// TwinCAT 3 PLC project PLC01
// ProgramVersion: 3.1.4024.0
// libraries:
//   Tc2_Standard, * (Beckhoff Automation GmbH)
//   Tc2_System, * (Beckhoff Automation GmbH)
//   Tc2_Utilities, * (Beckhoff Automation GmbH)
//   Tc3_Database, * (Beckhoff Automation GmbH)
//   Tc3_EventLogger, * (Beckhoff Automation GmbH)
//   Tc3_Module, * (Beckhoff Automation GmbH)
// project tree:
//   DUTs/ ST_Database.TcDUT
//   FBs/ FB_SQLMode_ExecuteCommandWithData.TcPOU, FB_SQLMode_ExecuteComandWithoutData.TcPOU, FB_SQLMode_ExecuteStoredProcedureWithoutData.TcPOU, FB_SQLMode_ExecuteStoredProcedureWithData.TcPOU
//   / PlcTask.TcTTO
//   POUs/ MAIN.TcPOU
//   POUs/PLC Mode/ PLC_Mode.TcPOU, PRG_CreateDatabasePlcMode.TcPOU, PRG_CreateTablePlcMode.TcPOU, PRG_DeleteRowDatabasePlcMode.TcPOU, PRG_ReadDatabasePlcMode.TcPOU, PRG_WriteDatabasePlcMode.TcPOU
//   POUs/SQL Mode/ PRG_CreateDatabaseSqlMode.TcPOU, PRG_CreateTableSqlMode.TcPOU, PRG_DeleteRowSqlMode.TcPOU, PRG_ReadDatabaseSqlMode.TcPOU, PRG_WriteDatabaseSqlMode.TcPOU, SQL_Mode.TcPOU
// real-time tasks:
//   TASK PlcTask: cycle T#10ms, priority 20, ADS port 350

CONFIGURATION PLC01
    RESOURCE PLC ON TwinCAT3
        TASK PlcTask(INTERVAL := T#10ms, PRIORITY := 20);
        PROGRAM MAIN WITH PlcTask : MAIN;
    END_RESOURCE
END_CONFIGURATION

// ---- DUTs/ST_Database.TcDUT
TYPE ST_Database :
STRUCT
	ID : T_ULARGE_INTEGER  ;	//IDENTITY
	Timestamp : DATE_AND_TIME ;	//TIMESTAMP
	recipe : STRING(51) ;		//NAME OF RECIPE
	parameter1 : LREAL ;		//PARAMETER 1
	parameter2 : LREAL ;		//PARAMETER 2
	parameter3 : LREAL ;		//PARAMETER 3
	parameter4 : LREAL ;		//PARAMETER 4
	parameter5 : LREAL ;		//PARAMETER 5
	parameter6 : LREAL ;		//PARAMETER 6
END_STRUCT
END_TYPE

// ---- POUs/MAIN.TcPOU
PROGRAM MAIN
VAR
END_VAR

PLC_Mode() ;

SQL_Mode();

END_PROGRAM

// ---- POUs/PLC Mode/PLC_Mode.TcPOU
PROGRAM PLC_Mode
VAR
END_VAR

PRG_CreateDatabasePlcMode();

PRG_CreateTablePlcMode();

PRG_DeleteRowDatabasePlcMode();

PRG_WriteDatabasePlcMode();

PRG_ReadDatabasePlcMode();

END_PROGRAM

// ---- POUs/PLC Mode/PRG_CreateDatabasePlcMode.TcPOU
PROGRAM PRG_CreateDatabasePlcMode
VAR
    fbPLCDBCreate : FB_PLCDBCreateEvt(sNetID := '', tTimeout := T#5S);
    stConfigDB    : T_DBConfig_MsSQL;
    hDBID         : UDINT ;
    tcMessage     : I_TcMessage;
	nState : INT ;	
	bCreateDatabase: BOOL;
	sMessage : STRING ;
END_VAR

stConfigDB.sProvider := 'SQLOLEDB' ;
stConfigDB.sServer:= 'DOUGLASC-NB01\SQLEXPRESS';
stConfigDB.sDatabase := 'MyDatabase123';
stConfigDB.bAuthentification := TRUE;
stConfigDB.sUserID := 'sa';
stConfigDB.sPassword := 'sa';

IF bCreateDatabase = TRUE THEN
	IF fbPLCDBCreate.Database(
		pDatabaseConfig:= ADR(stConfigDB),
		cbDatabaseConfig := SIZEOF(stConfigDB),
		bCreateXMLConfig := TRUE,
		pDBID := ADR(hDBID))
	THEN
		IF fbPLCDBCreate.bError THEN
			tcMessage := fbPLCDBCreate.ipTcResult;
			bCreateDatabase := FALSE ;
			sMessage := 'Error';
		ELSE
			bCreateDatabase := FALSE ;
			sMessage := 'OK';
		END_IF
	END_IF
END_IF

END_PROGRAM

// ---- POUs/PLC Mode/PRG_CreateTablePlcMode.TcPOU
PROGRAM PRG_CreateTablePlcMode
VAR
    fbPLCDBCreate	: FB_PLCDBCreateEvt(sNetID := '', tTimeout := T#5S);	//Bloco para criar a tabela
    ColumnInfo		: ARRAY [0..8] OF ST_ColumnInfo ;						//Estrutura com a tabela a ser criada
    tcMessage		: I_TcMessage;											//Variavel para tratamento das mensagens
	bCreateTable	: BOOL ; 												//Bit para criar tabela
	sError : STRING ;														//String com a mensagem de erro
END_VAR

(* Exemplos : 
ColumnInfo[0].sName := 'colBigInt';     ColumnInfo[0].eType := E_ColumnType.BigInt;     ColumnInfo[0].nLength := 8;     ColumnInfo[0].sProperty := 'IDENTITY(1,1)';
ColumnInfo[1].sName := 'colInteger';    ColumnInfo[1].eType := E_ColumnType.Integer;    ColumnInfo[1].nLength := 4;
ColumnInfo[2].sName := 'colSmallInt';   ColumnInfo[2].eType := E_ColumnType.SmallInt;   ColumnInfo[2].nLength := 2;
ColumnInfo[3].sName := 'colTinyInt';    ColumnInfo[3].eType := E_ColumnType.TinyInt;    ColumnInfo[3].nLength := 1;
ColumnInfo[4].sName := 'colBit';        ColumnInfo[4].eType := E_ColumnType.BIT_;       ColumnInfo[4].nLength := 1;
ColumnInfo[5].sName := 'colMoney';      ColumnInfo[5].eType := E_ColumnType.Money;      ColumnInfo[5].nLength := 8;
ColumnInfo[6].sName := 'colFloat';      ColumnInfo[6].eType := E_ColumnType.Float;      ColumnInfo[6].nLength := 8;
ColumnInfo[7].sName := 'colReal';       ColumnInfo[7].eType := E_ColumnType.REAL_;      ColumnInfo[7].nLength := 4;
ColumnInfo[8].sName := 'colDateTime';   ColumnInfo[8].eType := E_ColumnType.DateTime;   ColumnInfo[8].nLength := 4;
ColumnInfo[9].sName := 'colNText';      ColumnInfo[9].eType := E_ColumnType.NText;      ColumnInfo[9].nLength := 256;
ColumnInfo[10].sName := 'colNChar';     ColumnInfo[10].eType := E_ColumnType.NChar;     ColumnInfo[10].nLength := 10;
ColumnInfo[11].sName := 'colImage';     ColumnInfo[11].eType := E_ColumnType.Image;     ColumnInfo[11].nLength := 256;
ColumnInfo[12].sName := 'colNVarChar';  ColumnInfo[12].eType := E_ColumnType.NVarChar;  ColumnInfo[12].nLength := 50;
ColumnInfo[13].sName := 'colBinary';    ColumnInfo[13].eType := E_ColumnType.Binary;    ColumnInfo[13].nLength := 30;
ColumnInfo[14].sName := 'colVarBinary'; ColumnInfo[14].eType := E_ColumnType.VarBinary; ColumnInfo[14].nLength := 20;
*)

(* A criação das tabelas pode ser feita pelo código do PLC, mas também através da janela Sql Query Edition *)
(* Declaração da estrutura da tabela *)

ColumnInfo[0].sName := 'ID';     ColumnInfo[0].eType := E_ColumnType.BigInt;     ColumnInfo[0].nLength := 8;     ColumnInfo[0].sProperty := 'IDENTITY(1,1)';
ColumnInfo[1].sName := 'Timestamp';   ColumnInfo[1].eType := E_ColumnType.DateTime;   ColumnInfo[1].nLength := 4;
ColumnInfo[2].sName := 'recipe';  ColumnInfo[2].eType := E_ColumnType.NVarChar;  ColumnInfo[2].nLength := 50;
ColumnInfo[3].sName := 'parameter1';      ColumnInfo[3].eType := E_ColumnType.Float;      ColumnInfo[3].nLength := 8;
ColumnInfo[4].sName := 'parameter2';      ColumnInfo[4].eType := E_ColumnType.Float;      ColumnInfo[4].nLength := 8;
ColumnInfo[5].sName := 'parameter3';      ColumnInfo[5].eType := E_ColumnType.Float;      ColumnInfo[5].nLength := 8;
ColumnInfo[6].sName := 'parameter4';      ColumnInfo[6].eType := E_ColumnType.Float;      ColumnInfo[6].nLength := 8;
ColumnInfo[7].sName := 'parameter5';      ColumnInfo[7].eType := E_ColumnType.Float;      ColumnInfo[7].nLength := 8;
ColumnInfo[8].sName := 'parameter6';      ColumnInfo[8].eType := E_ColumnType.Float;      ColumnInfo[8].nLength := 8;

(* Para criar a tabela colocar a variavel bCreateTable em TRUE *)
(* To Create Table put the bCreateTable variable in TRUE *)
IF bCreateTable = TRUE THEN
	IF fbPLCDBCreate.Table(
		hDBID:= 1,
		sTableName:= 'TB_PLCMODE', 
		pTableCfg:= ADR(ColumnInfo), 
		cbTableCfg:= SIZEOF(ColumnInfo))
	THEN
		IF fbPLCDBCreate.bError THEN
			TcMessage:= fbPLCDBCreate.ipTcResult;
			sError := 'Erro'; 
		ELSE
			sError := 'OK';
		END_IF
	END_IF
	bCreateTable := FALSE ;	
END_IF

END_PROGRAM

// ---- POUs/PLC Mode/PRG_DeleteRowDatabasePlcMode.TcPOU
PROGRAM PRG_DeleteRowDatabasePlcMode
VAR
//Variáveis de conexão / Connection variables
	hDBID: UDINT := 1 ;							//DB ID
    sTableName: T_MaxString := 'TB_PLCMODE' ;	//Nome da Tabela / Table name

    fbPLCDBCmd		: FB_PLCDBCmdEvt(sNetID := '', tTimeout := T#5S);
    sCommandDelete  : STRING (1000);									//Comando SQL / SQL Command
    stParameter 	: ARRAY [1..1] OF ST_ExpParameter; 					//Parametros do comando SQL / Parameter SQL Command
    sRecipeName		: STRING(80) := 'recipe'; 							//Nome da receita a ser deletada / Recipe name to delete	
	bExecuteDelete 	: BOOL ;											//Executar delete / Execute delete	
	sMessageError	: STRING ;											//Mensagem de status / Status message
    tcMessageDelete	: I_TcMessage;										//
END_VAR

(***************************** CODE TO DELETE ONE ROW IN DATABASE             ***************************************)
(***************************** CODIGO PARA DELETAR UMA LINHA DO BANCO DE DADOS***************************************)

(* PARAMETER TO DELETE ONE RECIPE *)
(* PARAMETRO PARA DELETAR UMA RECEITA *)

stParameter[1].sParaName := 'sRecipeName';
stParameter[1].eParaType := E_ExpParameterType.STRING_;
stParameter[1].nParaSize := SIZEOF(sRecipeName);

(* SQL COMMAND TO DELETE A LINE THAT CONTAINS THE NAME DEFINED IN THE sRecipeName VARIABLE *)
(* COMANDO SQL PARA DELETAR UMA LINHA QUE CONTENHA O NOME DEFINIDO NA VARIAVEL sRecipeName *)
 sCommandDelete := 'DELETE FROM TB_PLCMODE WHERE recipe = {sRecipeName} ' ;
 
 
(* EXECUTE COMMAND TO DELETE THE ROW*)
(* EXECUTA COMANDO PARA DELETAR A LINHA *)
IF bExecuteDelete THEN

	IF fbPLCDBCmd.Execute(
		hDBID:= 1,
		pExpression:= ADR(sCommandDelete),
		cbExpression:= SIZEOF(sCommandDelete),
		pData:= ADR(sRecipeName),
		cbData:= SIZEOF(sRecipeName),
		pParameter:= ADR(stParameter),
		cbParameter:= SIZEOF(stParameter))				
	THEN	
		IF fbPLCDBCmd.bError THEN
			sMessageError := 'ERROR';
			bExecuteDelete := FALSE ;			
			tcMessageDelete := fbPLCDBCmd.ipTcResult;
		ELSE
			sMessageError := 'OK';
			bExecuteDelete := FALSE ;
		END_IF
	END_IF
END_IF

END_PROGRAM

// ---- POUs/PLC Mode/PRG_WriteDatabasePlcMode.TcPOU
PROGRAM PRG_WriteDatabasePlcMode
VAR
	hDBID: UDINT := 1 ;							//DB ID
    sTableName: T_MaxString := 'TB_PLCMODE' ;	//NOME DA TABELA / TABLE NAME / NOMBRE DA TABLA

//ESCREVER NO BANCO DE DADOS / WRITE DO DATABASE / ESCRIBIR EN LA BASE DE DATOS 
    fbPLCDBWrite    :	FB_PLCDBWriteEvt(sNetID := '', tTimeout := T#5S);//
    DataToDB 		:	ST_Database;									 //ESTRUTURA A ESCRITA NO BANCO / STRUCT TO SEND TO DATABASE
    ColumnNames     :	ARRAY[0..8] OF STRING(50);						 //ESTRUTURA COM O NOME DAS COLUNAS / STRUCT WITH COLLUNS NAME
    systime         :	GETSYSTEMTIME;									 //DATA E HORA DO  SISTEMA / DATE TIME OF SYSTEM
    currentTime     :	T_FILETIME;										 //
    tcMessage_Write :	I_TcMessage;									 //
	
	bWriteValues : BOOL ;	
	sMessage : STRING ;
	iRecipeNumerForTest : INT ;

END_VAR

//NOME DAS COLUNAS DA TABELA / NAME OF THE TABLE COLUMNS/
ColumnNames[0] := 'ID';
ColumnNames[1] := 'Timestamp';
ColumnNames[2] := 'recipe';
ColumnNames[3] := 'parameter1';
ColumnNames[4] := 'parameter2';
ColumnNames[5] := 'parameter3';
ColumnNames[6] := 'parameter4';
ColumnNames[7] := 'parameter5';
ColumnNames[8] := 'parameter6';

(* Logica de teste apenas para gerar dados para gravar no banco *)

systime(timeLoDw => currentTime.dwLowDateTime, timeHiDW => currentTime.dwHighDateTime );


(* SIMULATE VALUES TO WRITE TO DATABASE *)
IF bWriteValues THEN
	
//Simulacao de valores 
	DataToDB.Timestamp  := FILETIME_TO_DT(currentTime);;
	DataToDB.recipe     := CONCAT ('recipe', TO_STRING(iRecipeNumerForTest)) ;
	DataToDB.parameter1 := DataToDB.parameter1 + 10;
	DataToDB.parameter2 := DataToDB.parameter2 + 10;
	DataToDB.parameter3	:= DataToDB.parameter3 + 10 ;
	DataToDB.parameter4 := DataToDB.parameter4 + 10 ;
	DataToDB.parameter5 := DataToDB.parameter5 + 10 ;
	DataToDB.parameter6 := DataToDB.parameter6 + 10 ;

	
END_IF
	
/////////////////////////////// Chamada da função de escrita
IF bWriteValues THEN
	IF fbPLCDBWrite.WriteStruct(
		hDBID:= hDBID, 
		sTableName:= sTableName, 
		pRecord:= ADR(DataToDB), 
		cbRecord:= SIZEOF(DataToDB), 
		pColumnNames:= ADR(ColumnNames) , 
		cbColumnNames:= SIZEOF(ColumnNames))
	THEN
		IF fbPLCDBWrite.bError THEN
			tcMessage_Write := fbPLCDBWrite.ipTcResult;
			sMessage := 'ERROR';
			bWriteValues := FALSE ;	 
		ELSE
			sMessage := 'OK';
			bWriteValues := FALSE ;	 
		END_IF
	END_IF
END_IF

END_PROGRAM

// ---- POUs/PLC Mode/PRG_ReadDatabasePlcMode.TcPOU
PROGRAM PRG_ReadDatabasePlcMode
VAR
//Variáveis gerais
	hDBID: UDINT := 1 ;							//DB ID - Ver banco no database server
    sTableName: T_MaxString := 'TB_PLCMODE' ;	//Nome da Tabela

//Ler dados da tabela comando SELECT
    fbPLCDBCmd   : FB_PLCDBCmdEvt(sNetID := '', tTimeout := T#5S);	//Bloco para leitura dos dados via comando SQL
    sCommandSql  : STRING (1000); 									//Comando SQL	
    stParametros : ARRAY [0..0] OF ST_ExpParameter; 				//Parametros usado no filtro SQL	
    sReceita : STRING ; 											//Parametros usado no filtro SQL	
	bCommandSelect: BOOL ;											//
	sMenssageError : STRING ; 										//
    nRecords : BYTE ;												//
	DBToData : ARRAY [0..9] OF ST_Database;							//
	
//Ler dados da tabela usando o bloco Read Struct
    fbPLCDBRead    	: FB_PLCDBReadEvt (sNetID := '', tTimeout := T#5S);	//Bloco para leitura do banco de dados sem filtro
    DBtoPLC 		: ARRAY [0..10] OF ST_Database;						//Dados recebidos do banco de dados
    ColumnNamesRead :  ARRAY[0..8] OF STRING(50);						//Lista com os nomes das colunas do banco de dados
    tcMessage      	: I_TcMessage;										//Estrutura para diagnosticos
	bReadStruct 	: BOOL ;											//Comando para ler banco de dados sem filtro
	sMenssageError1 	: STRING ; 										//Mensagem de erro

END_VAR


(* Nome das colunas / Columns Name *)
ColumnNamesRead[0] := 'ID' ;
ColumnNamesRead[1] := 'Timestamp';
ColumnNamesRead[2] := 'recipe';
ColumnNamesRead[3] := 'parameter1';
ColumnNamesRead[4] := 'parameter2';
ColumnNamesRead[5] := 'parameter3';
ColumnNamesRead[6] := 'parameter4';
ColumnNamesRead[7] := 'parameter5';
ColumnNamesRead[8] := 'parameter6';

(* Parametro: nome da receita a ser retornada*)
(* Parameter: name of the recipe to be returned*)

stParametros[0].sParaName := 'sReceita';
stParametros[0].eParaType := E_ExpParameterType.STRING_;
stParametros[0].nParaSize := SIZEOF(sReceita);

//////////////////// Comando SELECT////////////////////////

sCommandSql := 'SELECT ID, Timestamp, recipe, parameter1, parameter2, parameter3, parameter4, parameter5, parameter6 FROM TB_PLCMODE  WHERE recipe = {sReceita}';
   
IF bCommandSelect THEN			    
			   
	IF fbPLCDBCmd.ExecuteDataReturn(
		hDBID:= hDBID, 
		pExpression:= ADR(sCommandSql), 
		cbExpression:= SIZEOF(sCommandSql), 
		pData:= ADR(sReceita), 
		cbData:= SIZEOF(sReceita), 
		pParameter:= ADR(stParametros), 
		cbParameter:= SIZEOF(stParametros),
		nStartIndex:= 0, 
		nRecordCount:= 1, 
		pReturnData:= ADR(DBToData), 
		cbReturnData:= SIZEOF(DBToData), 
		pRecords:= ADR(nRecords)) 
	THEN
		 //Se nao estiver em erro ou ocupado desliga o bit
		IF fbPLCDBCmd.bError THEN
			sMenssageError := 'ERROR'; 
			bCommandSelect := FALSE ;			
		ELSE
			sMenssageError := 'OK'; 
			bCommandSelect := FALSE ;			
		END_IF
	END_IF
END_IF
	
		
	
(*****************************************************************************************************)	
(* FB para ler as 100 primeiras linhas da tabela *)
(*FB to read the first 100 rows of the table*)
	
IF bReadStruct THEN	 
	IF fbPLCDBRead.ReadStruct(
		hDBID:= 1, 
		sTableName:= 'TB_Recipes', 
		pColumnNames:= ADR(ColumnNamesRead), 
		cbColumnNames:= SIZEOF(ColumnNamesRead), 
		sOrderByColumn:= ColumnNamesRead[0], 
		eOrderType:= E_OrderType.ASC, 
		nStartIndex:= 0, 
		nRecordCount:= 100, 
		pData:= ADR(DBtoPLC), 
		cbData:= SIZEOF(DBtoPLC))
THEN
		IF fbPLCDBRead.bError THEN
			tcMessage:= fbPLCDBRead.ipTcResult;
			sMenssageError1 := 'ERROR'; 
			bReadStruct := FALSE ;			
		ELSE
			sMenssageError1 := 'OK'; 
			bReadStruct := FALSE ;
		END_IF
	END_IF	
END_IF

END_PROGRAM

// ---- POUs/SQL Mode/SQL_Mode.TcPOU
PROGRAM SQL_Mode
VAR
END_VAR

PRG_CreateTableSqlMode();

PRG_DeleteRowSqlMode();

PRG_ReadDatabaseSqlMode();

PRG_WriteDatabaseSqlMode();

PRG_CreateDatabaseSqlMode();

END_PROGRAM

// ---- POUs/SQL Mode/PRG_CreateTableSqlMode.TcPOU
PROGRAM PRG_CreateTableSqlMode
VAR
(* CRIAR TABELA / CREATE TABLE / CREAR TABLA *)	
	fbCreateTable : FB_SQLMode_ExecuteComandWithoutData ;
	bCreateDatabase : BOOL ;
	bDatabaseCreated : BOOL ;
	sSqlCmdCreateTable : STRING(512) ;
	sError : STRING ;
END_VAR

(***************** CRIAR TABELA / CREATE TABLE / CREAR TABLA **********************)

sSqlCmdCreateTable := 'CREATE TABLE [TB_SQLMODE] ([ID] bigint IDENTITY(1,1), [Timestamp] datetime,
[recipe] varchar(50), [parameter1] float, [parameter2] float, [parameter3] float, [parameter4] float,
[parameter5] float, [parameter6] float)';

fbCreateTable(bExecute:= bCreateDatabase, 
			  hDBID:= 1, 
			  sCommandSql:= sSqlCmdCreateTable, 
			  bCommandOk=> bDatabaseCreated,
			  sError => sError);

END_PROGRAM

// ---- FBs/FB_SQLMode_ExecuteComandWithoutData.TcPOU
FUNCTION_BLOCK FB_SQLMode_ExecuteComandWithoutData
VAR_INPUT
	bExecute : BOOL ;
	hDBID : UINT ;
	sCommandSql : STRING(512) ;
END_VAR
VAR_OUTPUT
	bCommandOk : BOOL ;
	sError : STRING ;
END_VAR
VAR
	fbSqlDatabase : FB_SQLDatabaseEvt(sNetID := '', tTimeout := T#5S);
	fbSqlCommand : FB_SQLCommandEvt(sNetID := '', tTimeout := T#5S) ;
    tcMessage    : I_TcMessage;	
	nState : INT ;
	fbPulse : R_TRIG ;
END_VAR

fbPulse(CLK:= bExecute, Q=> );

IF fbPulse.Q THEN
	nState := 1 ;
END_IF

CASE nState OF
		
	0: (* Iddle *)
	;
	
	1:
	bCommandOk := FALSE ;
	sError := '';
	nState := 10; 
	
	10: (* Connect to Database *)
	
	IF fbSqlDatabase.Connect(hDBID) THEN
		IF fbSqlDatabase.bError THEN
			nState := 250; 
        	tcMessage := fbSqlDatabase.ipTcResult;			
		ELSE
			nState := 20; 
		END_IF
	END_IF
	
	20:	(* Create Command *)
	
	IF fbSqlDatabase.CreateCmd(ADR(fbSqlCommand)) THEN
		IF fbSqlDatabase.bError THEN
			nState := 251; 
		ELSE
			nState := 30; 
		END_IF
	END_IF	
	
	30:  (* Execute Command *)
	
	IF fbSqlCommand.Execute(pSQLCmd:= ADR(sCommandSql), cbSQLCmd:= SIZEOF(sCommandSql)) THEN
		IF fbSQLCommand.bError THEN
			nState := 252; 
        	tcMessage := fbSQLCommand.ipTcResult;			
			bCommandOk := FALSE ;			
		ELSE
			nState := 40; 
			bCommandOk := TRUE ;
			sError := 'Comando OK';			
		END_IF
	END_IF	
	

	40:  (* Desconectar *)
	
	IF fbSqlDatabase.Disconnect() THEN
		IF fbSqlDatabase.bError THEN
			nState := 253;
		ELSE
			nState := 0;
   		END_IF
	END_IF

250: //Error step 10;
	sError := 'Erro no bloco Connect';
	nState := 40 ;

251: //Error step 20 ;
	sError := 'Erro no bloco Create Command';
	nState := 40 ;
252: //Error step 30 ;
	sError := 'Erro no bloco Execute Command';
	nState := 40 ;
253: //Error step 40 ;
	sError := 'Erro no bloco Disconect';
	nState := 40 ;
	
END_CASE

END_FUNCTION_BLOCK

// ---- POUs/SQL Mode/PRG_DeleteRowSqlMode.TcPOU
PROGRAM PRG_DeleteRowSqlMode
VAR
END_VAR

END_PROGRAM

// ---- POUs/SQL Mode/PRG_ReadDatabaseSqlMode.TcPOU
PROGRAM PRG_ReadDatabaseSqlMode
VAR
(* LER DO BANCO / READ FROM DATABASE / LEER DATABASE *)	
	fbReadSqlMode : FB_SQLMode_ExecuteCommandWithData ;
	bReadDatabase : BOOL ;	
	bWriteOk : BOOL ;	
	sSqlCmdReadTable : STRING(512) ;	
	sError : STRING ;
    aReadStruct : ARRAY[1..10] OF ST_Database;	
	
END_VAR


sSqlCmdReadTable :='SELECT [ID], [Timestamp], [recipe], [parameter1], [parameter2], [parameter3], 
[parameter4], [parameter5], [parameter6] FROM [dbo].[TB_SQLMODE] ';

fbReadSqlMode(
	bExecute:= bReadDatabase, 
	hDBID:= 1, 
	sCommandSql:= sSqlCmdReadTable, 
	bCommandOk=> , 
	sError=> sError, 
	aReadStruct=> aReadStruct);

END_PROGRAM

// ---- FBs/FB_SQLMode_ExecuteCommandWithData.TcPOU
FUNCTION_BLOCK FB_SQLMode_ExecuteCommandWithData
VAR_INPUT
	bExecute : BOOL ;
	hDBID : UINT ;
	sCommandSql : STRING(512) ;
END_VAR
VAR_OUTPUT
	bCommandOk : BOOL ;
	sError : STRING ;
    aReadStruct : ARRAY[1..10] OF ST_Database;	
END_VAR
VAR
    fbSqlDatabase : FB_SQLDatabaseEvt(sNetID := '', tTimeout := T#5S);
	fbSqlCommand : FB_SQLCommandEvt(sNetID := '', tTimeout := T#5S) ;
    tcMessage    : I_TcMessage;	
    fbSqlResult : FB_SQLResultEvt(sNetID:='', tTimeout    := T#5S); 	
	nState : INT ;
	fbPulse : R_TRIG ;
	bSqlResult : BOOL ;
	rParameter_old : REAL ;
END_VAR

fbPulse(CLK:= bExecute, Q=> );

IF fbPulse.Q THEN
	nState := 1;		
END_IF

CASE nState OF
		
	0: ; //PARADO / IDLE / INTERRUMPIDO
		
	1: //INICIALIZA VARIAVEIS / START VARIABLES /  INICIALIZAR VARIABLES
		bCommandOk := FALSE ;
		sError := '' ;	
		rParameter_old := 0 ;			

		IF fbSqlDatabase.Disconnect() THEN
			IF fbSqlDatabase.bError THEN
				nState := 255;
			ELSE
				nState := 10;
			END_IF
		END_IF
	
	10: //ABRIR CONEXAO / OPEN CONECTION / CONEXION ABIERTA
	
		IF fbSqlDatabase.Connect(hDBID:= hDBID) THEN
			IF fbSqlDatabase.bError THEN
				nState := 210; 
			ELSE
				nState := 20; 
			END_IF
		END_IF
	
	20: //CRIAR COMANDO / CREATE COMMAND / CREAR COMANDO
	
		IF fbSqlDatabase.CreateCmd(ADR(fbSqlCommand)) THEN
			IF fbSqlDatabase.bError THEN
				nState := 220; 			
			ELSE
				nState := 30; 
			END_IF
		END_IF	
		
	30: //EXECUTA COMANDO / EXCUTE COMMAND / EJECUTAR COMANDO
	
		IF fbSqlCommand.ExecuteDataReturn(pSQLCmd:= ADR(sCommandSql), cbSQLCmd:= SIZEOF(sCommandSql), pSQLDBResult:= ADR(fbSqlResult)) THEN
			IF fbSQLCommand.bError THEN
				nState := 230; 				
				tcMessage := fbSQLCommand.ipTcResult;
			ELSE
				nState := 40; 
			END_IF
		END_IF
				
				
	40: //RECEBE OS DADOS / RECEIVE DATA / RECIBIR LOS DATOS
		bSqlResult := 	fbSqlResult.Read(nStartIndex:= 1,nRecordCount:= 10, pData:= ADR(aReadStruct), cbData:= SIZEOF(aReadStruct), bWithVerifying:= FALSE, bDataRelease:= TRUE) ;

		IF fbSqlResult.bError THEN
			nState := 240 ;
		ELSE
			nState := 50; 
		END_IF		

	
	50: //EXTRAI OS VALORES DO BUFFER / EXTRACT DATA FROM BUFFER
		fbSqlResult.Release();
			IF fbSqlResult.bError THEN
				nState := 250; 
			ELSE
				nState := 55; 
				sError := 'OK' ;
				bCommandOk := TRUE ;				
			END_IF
			
	55: //VERIFICA SE FORAM RETORNADOS DADOS / CHECK DATA RETURN		
		IF aReadStruct[1].parameter1 <>	rParameter_old THEN
			rParameter_old := aReadStruct[1].parameter1 ;
			nState := 60;
		ELSE
			nState := 20; 			 			
		END_IF
			
	60: //DESCONECTAR DO BANCO / DATABASE DISCONECT
		IF fbSqlDatabase.Disconnect() THEN
			IF fbSqlDatabase.bError THEN
				nState := 255;
			ELSE
				nState := 0;			
			END_IF
		END_IF
		
	210 : 
		sError := 'Error Connect' ;
		nState := 60;		
		bCommandOk := FALSE ;	
	220 : 
		sError := 'Error Create Command' ;	
		nState := 60;	
		bCommandOk := FALSE ;			
	230: 
		sError := 'Error Execute Command' ;	
		nState := 60;	
		bCommandOk := FALSE ;			
	240: 
		sError := 'Error Read' ;			
		nState := 60;	
		
	250:
		sError := 'Error Release' ;		
		nState := 60;	
		bCommandOk := FALSE ;			
	260: 				
		sError := 'Error Disconect' ;	
		nState := 60;	
		bCommandOk := FALSE ;				
END_CASE

END_FUNCTION_BLOCK

// ---- POUs/SQL Mode/PRG_WriteDatabaseSqlMode.TcPOU
PROGRAM PRG_WriteDatabaseSqlMode
VAR
(* ESCREVER NO BANCO / WRITE TO DATABASE / ESCRIBIR EN LA DATABASE *)	
	fbWriteSqlMode : FB_SQLMode_ExecuteComandWithoutData ;
	bWriteDatabase : BOOL ;	
	bWriteOk : BOOL ;	
	sSqlCmdWriteTable : STRING(512) ;	
	sError : STRING ;	
	
    systime     : GETSYSTEMTIME; //DATA E HORA DO  SISTEMA / DATE TIME OF SYSTEM	
    currentTime : T_FILETIME;	 //	
	sTimestamp : STRING ;
	sRecipeName : STRING ;
	sParameter1 : STRING ;
	sParameter2 : STRING ;
	sParameter3 : STRING ;
	sParameter4 : STRING ;
	sParameter5 : STRING ;
	sParameter6 : STRING ;	
	
	dtTimestamp : DATE_AND_TIME;
	iRecipeNumerForTest : INT ;
	rParameter1 : REAL ;
	rParameter2 : REAL ;
	rParameter3 : REAL ;
	rParameter4 : REAL ;
	rParameter5 : REAL ;
	rParameter6 : REAL ;	
	
	fbPulse : F_TRIG ;
END_VAR


//SIMULA VALORES
systime(timeLoDw => currentTime.dwLowDateTime, timeHiDW => currentTime.dwHighDateTime );

fbPulse(CLK:= bWriteDatabase, Q=> );

IF fbPulse.Q THEN
	dtTimestamp  := fILETIME_TO_DT(currentTime);
	iRecipeNumerForTest := iRecipeNumerForTest + 1 ;
	rParameter1 := rParameter1 + 10;
	rParameter2 := rParameter2 + 10;
	rParameter3	:= rParameter3 + 10;
	rParameter4 := rParameter4 + 10;
	rParameter5 := rParameter5 + 10;
	rParameter6 := rParameter6 + 10;

END_IF

//CONVERTE NUMEROS SIMULADOS PARA STRING / CONVERT SIMULATE VALUES TO STRING
	sTimestamp  := TO_STRING(dtTimestamp);
	sRecipeName := CONCAT ('recipe', TO_STRING(iRecipeNumerForTest)) ;
	sParameter1 := TO_STRING(rParameter1);
	sParameter2 := TO_STRING(rParameter2);
	sParameter3	:= TO_STRING(rParameter3);
	sParameter4 := TO_STRING(rParameter4);
	sParameter5 := TO_STRING(rParameter5);
	sParameter6 := TO_STRING(rParameter6);




//COMANDO SQL / SQL COMMAND / 

sTimestamp := DELETE(sTimestamp, 3, 1) ; 
sTimestamp := REPLACE(sTimestamp, ' ', 1, 11) ; 
sSqlCmdWriteTable := CONCAT ('INSERT INTO [dbo].[TB_SQLMODE] ( [Timestamp], [recipe], [parameter1], [parameter2], [parameter3], [parameter4], [parameter5], [parameter6]) VALUES ( $'', sTimestamp) ;
sSqlCmdWriteTable := CONCAT (sSqlCmdWriteTable, '$', $'') ;
sSqlCmdWriteTable := CONCAT (sSqlCmdWriteTable, sRecipeName) ;
sSqlCmdWriteTable := CONCAT (sSqlCmdWriteTable, '$' , ') ;
sSqlCmdWriteTable := CONCAT (sSqlCmdWriteTable, sParameter1) ;
sSqlCmdWriteTable := CONCAT (sSqlCmdWriteTable, ', ') ;
sSqlCmdWriteTable := CONCAT (sSqlCmdWriteTable, sParameter2) ;
sSqlCmdWriteTable := CONCAT (sSqlCmdWriteTable, ', ') ;
sSqlCmdWriteTable := CONCAT (sSqlCmdWriteTable, sParameter3) ;
sSqlCmdWriteTable := CONCAT (sSqlCmdWriteTable, ', ') ;
sSqlCmdWriteTable := CONCAT (sSqlCmdWriteTable, sParameter4) ;
sSqlCmdWriteTable := CONCAT (sSqlCmdWriteTable, ', ') ;
sSqlCmdWriteTable := CONCAT (sSqlCmdWriteTable, sParameter5) ;
sSqlCmdWriteTable := CONCAT (sSqlCmdWriteTable, ', ') ;
sSqlCmdWriteTable := CONCAT (sSqlCmdWriteTable, sParameter6) ;
sSqlCmdWriteTable := CONCAT (sSqlCmdWriteTable, ' )') ;

//sSqlCmdWriteTable := 'INSERT INTO [dbo].[TB_SQLMODE] ( [Timestamp], [recipe], [parameter1], [parameter2], [parameter3], [parameter4], [parameter5], [parameter6]) VALUES ( $'2023-07-26 15:41:02$', $'recipe3$', 1.3, 2.3, 3.3, 4.3, 5.3, 6.3) ';


// FUNCTION BLOCK TO WRITE
fbWriteSqlMode(
	bExecute:= bWriteDatabase, 
	hDBID:= 1, 
	sCommandSql:= sSqlCmdWriteTable, 
	bCommandOk=> bWriteOk, 
	sError=> sError );
	
IF fbWriteSqlMode.bCommandOk THEN
	bWriteDatabase := FALSE ;
END_IF

END_PROGRAM

// ---- POUs/SQL Mode/PRG_CreateDatabaseSqlMode.TcPOU
PROGRAM PRG_CreateDatabaseSqlMode
VAR
(* CRIAR TABELA / CREATE TABLE / CREAR TABLA *)	
	fbCreateDatabase : FB_SQLMode_ExecuteComandWithoutData ;
	bCreateDatabase : BOOL ;
	bDatabaseCreated : BOOL ;
	sSqlCmdCreateDatabse : STRING(512) ;
	sError : STRING ;	
END_VAR

sSqlCmdCreateDatabse := 'CREATE DATABASE NomeDoBancoDeDados;';

fbCreateDatabase(bExecute:= bCreateDatabase, 
			  hDBID:= 1, 
			  sCommandSql:= sSqlCmdCreateDatabse, 
			  bCommandOk=> bDatabaseCreated,
			  sError => sError);

END_PROGRAM

// ---- FBs/FB_SQLMode_ExecuteStoredProcedureWithoutData.TcPOU
FUNCTION_BLOCK FB_SQLMode_ExecuteStoredProcedureWithoutData
VAR_INPUT
	bExecute : BOOL ;
	hDBID : UINT ;
	sCommandSql : STRING(512) ;	
END_VAR
VAR_OUTPUT
	bCommandOk : BOOL ;
	sError : STRING ;	
END_VAR
VAR
	fbSqlDatabase : FB_SQLDatabaseEvt(sNetID := '', tTimeout := T#5S);	
    fbSQLStoredProcedure : FB_SQLStoredProcedureEvt(sNetID:='', tTimeout    := T#5S);	
    ParaInfo        : ST_SQLSPParameter; 
	
    tcMessage    : I_TcMessage;	
	nState : INT ;
	fbPulse : R_TRIG ;	
	ID: BYTE;
END_VAR

fbPulse(CLK:= bExecute, Q=> );

IF fbPulse.Q THEN
	nState := 1 ;
END_IF

CASE nState OF
		
	0: (* Iddle *)
	;
	
	1:
	bCommandOk := FALSE ;
	sError := '';
	nState := 10; 
	
	10: (* Connect to Database *)
	
	IF fbSqlDatabase.Connect(hDBID) THEN
		IF fbSqlDatabase.bError THEN
			nState := 250; 
        	tcMessage := fbSqlDatabase.ipTcResult;			
		ELSE
			nState := 20; 
		END_IF
	END_IF
	
	20:	(* Create Command *)
	ParaInfo.sParameterName     := '@Customer_ID';
	ParaInfo.eParameterType     := E_SPParameterType.Input;
	ParaInfo.eParameterDataType := E_ColumnType.BigInt;
	ParaInfo.nParameterSize     := 8;
	
	IF fbSQLDatabase.CreateSP('dbo.SP_GetCustomerPositions', ADR(ParaInfo), SIZEOF(ParaInfo), ADR(fbSQLStoredProcedure)) THEN
		IF fbSQLDatabase.bError THEN
			nState:=255;
		ELSE
			nState:= nState+1;
		END_IF
	END_IF
	
	
	
	30:
	
	IF fbSQLStoredProcedure.Execute(pParameterStrc := ADR(ID) , cbParameterStrc:= SIZEOF(ID)) THEN
		IF fbSQLStoredProcedure.bError THEN
			tcMessage := fbSQLStoredProcedure.ipTcResult;
			nState := 255;
		ELSE
			nState := nState+1;
		END_IF
	END_IF

END_FUNCTION_BLOCK

// ---- FBs/FB_SQLMode_ExecuteStoredProcedureWithData.TcPOU
FUNCTION_BLOCK FB_SQLMode_ExecuteStoredProcedureWithData
VAR_INPUT
END_VAR
VAR_OUTPUT
END_VAR
VAR
END_VAR

END_FUNCTION_BLOCK
